PROGRAM MAIN_Services
VAR
END_VAR

END_PROGRAM

(* stored: Version 1.1.0.1, ProductVersion 3.1.4024.15
   POU MAIN_Services: Id {3af486fa-0c2d-4875-b9ea-bc50deddc50f}, SpecialFunc None *)
